(* PLC project Unnamed, Unknown Unnamed 1 *)
(* stored: creationDateTime 2025-11-02T15:09:55, modificationDateTime 2025-11-02T15:31:46 *)

FUNCTION_BLOCK TrafficLightSequence
  VAR_OUTPUT
    Sequence : INT := 1;
  END_VAR
  VAR
    StepTime : TIME := T#3s;
    TON0 : TON;
    TON1 : TON;
    TON2 : TON;
  END_VAR

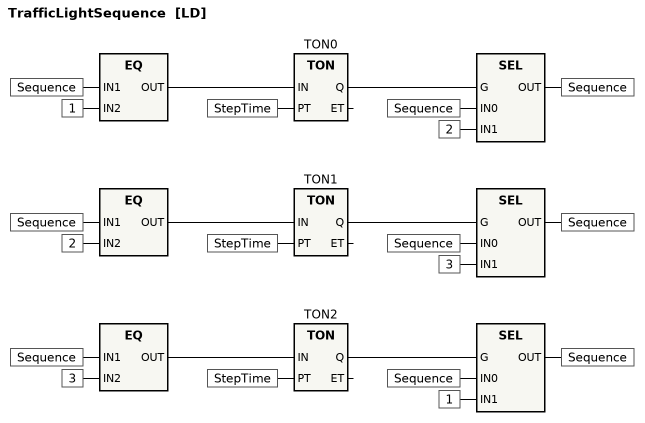
(* LD diagram, written out as Structured Text *)
TON0(IN := Sequence = 1, PT := StepTime);
Sequence := SEL(TON0.Q, Sequence, 2);
TON1(IN := Sequence = 2, PT := StepTime);
Sequence := SEL(TON1.Q, Sequence, 3);
TON2(IN := Sequence = 3, PT := StepTime);
Sequence := SEL(TON2.Q, Sequence, 1);
END_FUNCTION_BLOCK

PROGRAM TrafficLightControls
  VAR
    L_Red : BOOL := False;
    L_Yellow : BOOL := False;
    L_Green : BOOL := False;
    F_Sequence : INT;
    TrafficLightSequence0 : TrafficLightSequence;
  END_VAR

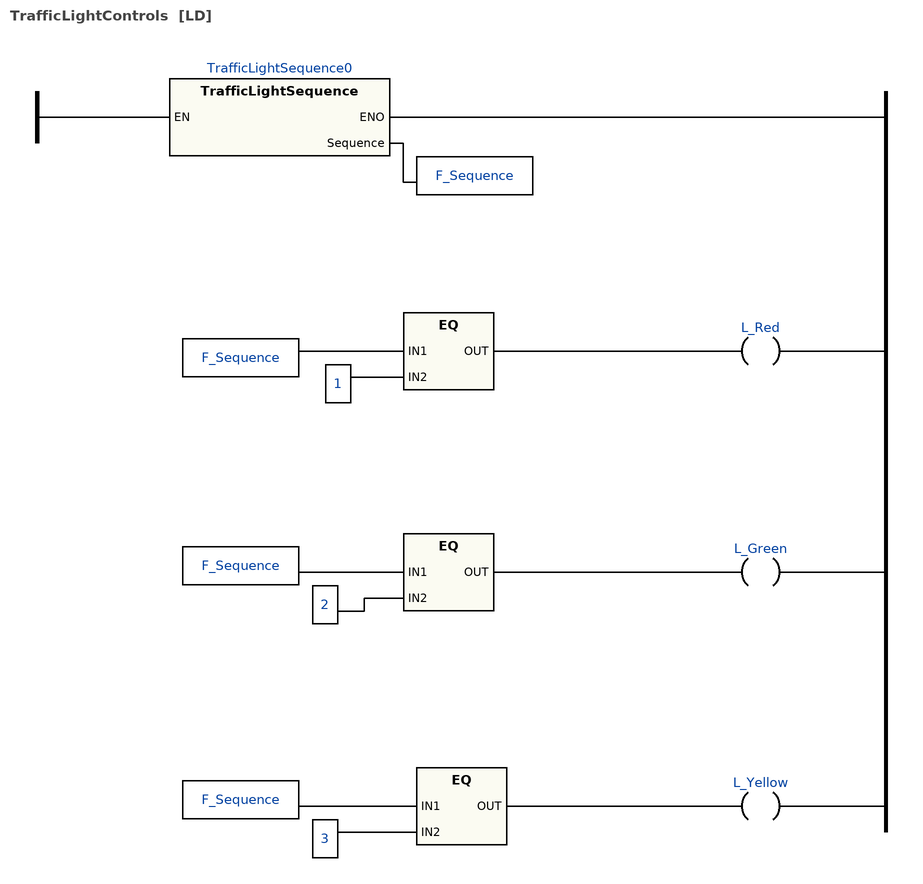
(* LD diagram, written out as Structured Text *)
TrafficLightSequence0();
F_Sequence := TrafficLightSequence0.Sequence;
L_Red := F_Sequence = 1;
L_Green := F_Sequence = 2;
L_Yellow := F_Sequence = 3;
END_PROGRAM

CONFIGURATION Config0
  RESOURCE Res0 ON PLC
    TASK task0(INTERVAL := T#20ms, PRIORITY := 0);
    PROGRAM instance0 WITH task0 : TrafficLightControls;
  END_RESOURCE
END_CONFIGURATION
